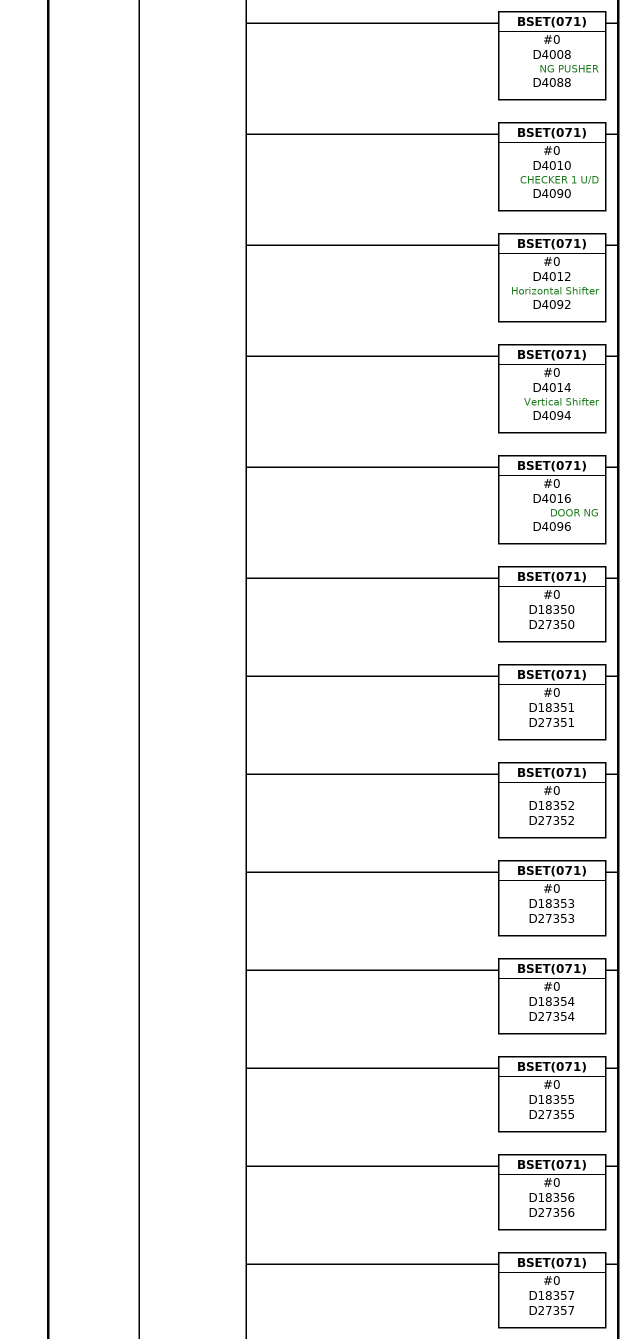
; [picture p48: Main_Control / Record, rungs 0-0]

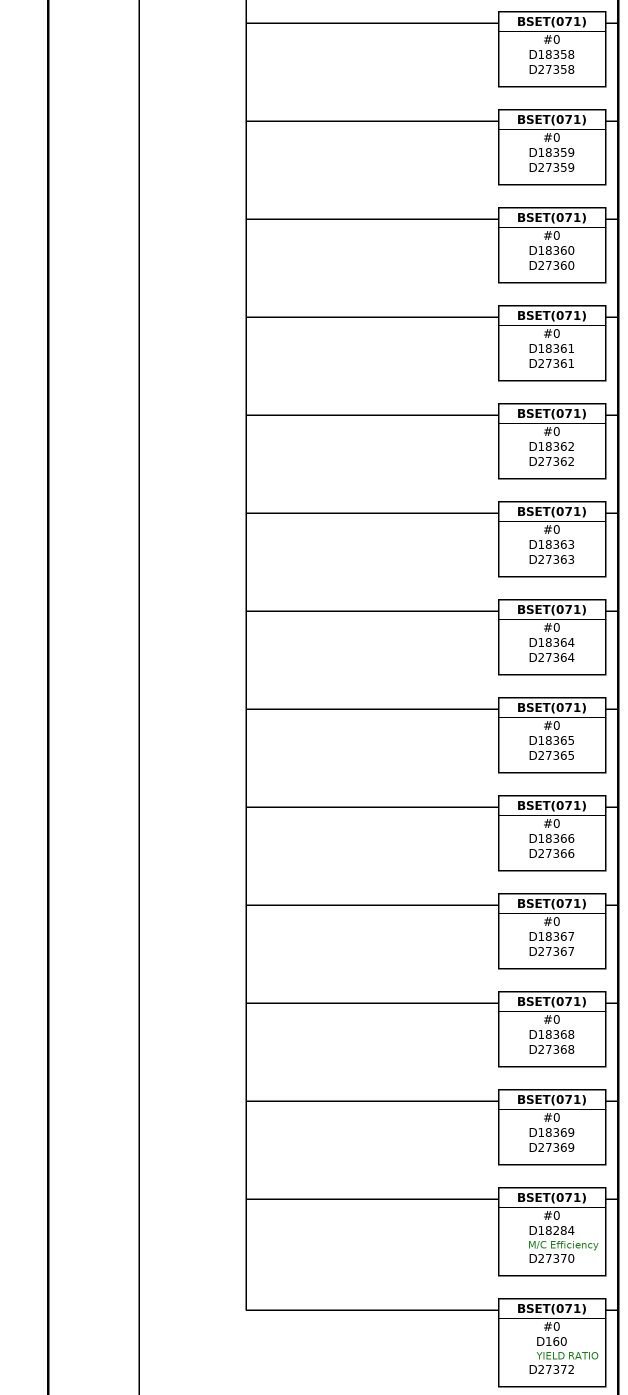

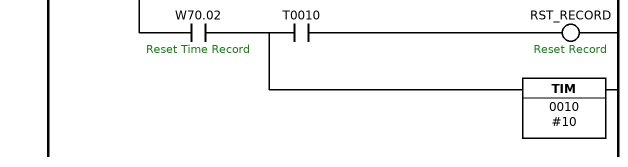
; rung 0: RESET MAIN RECORD
LD ON  ; ALWAYS ON
OUT TR0
@AND RST_RECORD  ; Reset Record
BSET(071) #0 D21300 D21399  ; OUTPUT OK
BSET(071) #0 D18251 D19299  ; M/C Cycle Time, $?St$Bk?_#[6] / $?St$Bk?_#[6]
BSET(071) #0 D19900 D19999  ; Auto Run (second), $?St$Bk?_#[7] / $?St$Bk?_#[7]
BSET(071) #0 D21100 D21199  ; STOP TIME (second)
BSET(071) #0 D21200 D21299  ; ALARM TIME (second)
BSET(071) #0 D18271 D18371  ; Input
BSET(071) #0 D20000 D20099  ; Total Alarm
BSET(071) #0 D4000 D4080  ; OVERLOAD
BSET(071) #0 D4002 D4082  ; STOPPER
BSET(071) #0 D4004 D4084  ; STOPPER CHECKER 1
BSET(071) #0 D4006 D4086  ; STOPPER CHECKER 2
BSET(071) #0 D4008 D4088  ; NG PUSHER
BSET(071) #0 D4010 D4090  ; CHECKER 1 U/D
BSET(071) #0 D4012 D4092  ; Horizontal Shifter
BSET(071) #0 D4014 D4094  ; Vertical Shifter
BSET(071) #0 D4016 D4096  ; DOOR NG
BSET(071) #0 D18350 D27350
BSET(071) #0 D18351 D27351
BSET(071) #0 D18352 D27352
BSET(071) #0 D18353 D27353
BSET(071) #0 D18354 D27354
BSET(071) #0 D18355 D27355
BSET(071) #0 D18356 D27356
BSET(071) #0 D18357 D27357
BSET(071) #0 D18358 D27358
BSET(071) #0 D18359 D27359
BSET(071) #0 D18360 D27360
BSET(071) #0 D18361 D27361
BSET(071) #0 D18362 D27362
BSET(071) #0 D18363 D27363
BSET(071) #0 D18364 D27364
BSET(071) #0 D18365 D27365
BSET(071) #0 D18366 D27366
BSET(071) #0 D18367 D27367
BSET(071) #0 D18368 D27368
BSET(071) #0 D18369 D27369
BSET(071) #0 D18284 D27370  ; M/C Efficiency
BSET(071) #0 D160 D27372  ; YIELD RATIO
LD TR0
AND W70.02  ; Reset Time Record
OUT TR0
AND T0010
OUT RST_RECORD  ; Reset Record
LD TR0
TIM 0010 #10

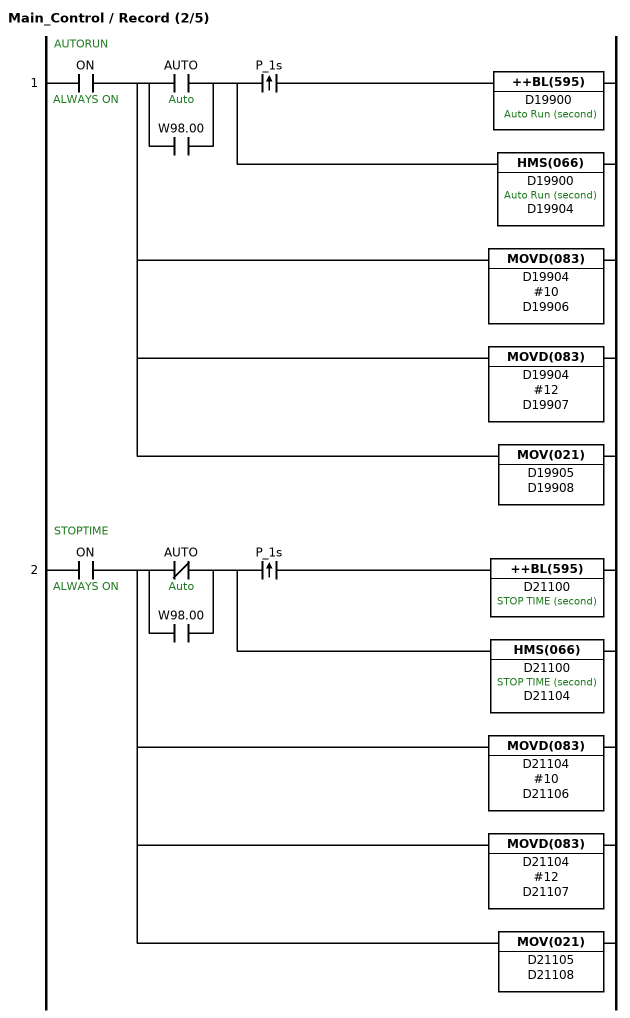
; rung 1: AUTORUN
LD ON  ; ALWAYS ON
OUT TR0
LD AUTO  ; Auto
OR W98.00
ANDLD
OUT TR1
@AND P_1s
++BL(595) D19900  ; Auto Run (second)
LD TR1
HMS(066) D19900 D19904  ; Auto Run (second)
LD TR0
MOVD(083) D19904 #10 D19906
MOVD(083) D19904 #12 D19907
MOV(021) D19905 D19908
; rung 2: STOPTIME
LD ON  ; ALWAYS ON
OUT TR0
LDNOT AUTO  ; Auto
OR W98.00
ANDLD
OUT TR1
@AND P_1s
++BL(595) D21100  ; STOP TIME (second)
LD TR1
HMS(066) D21100 D21104  ; STOP TIME (second)
LD TR0
MOVD(083) D21104 #10 D21106
MOVD(083) D21104 #12 D21107
MOV(021) D21105 D21108

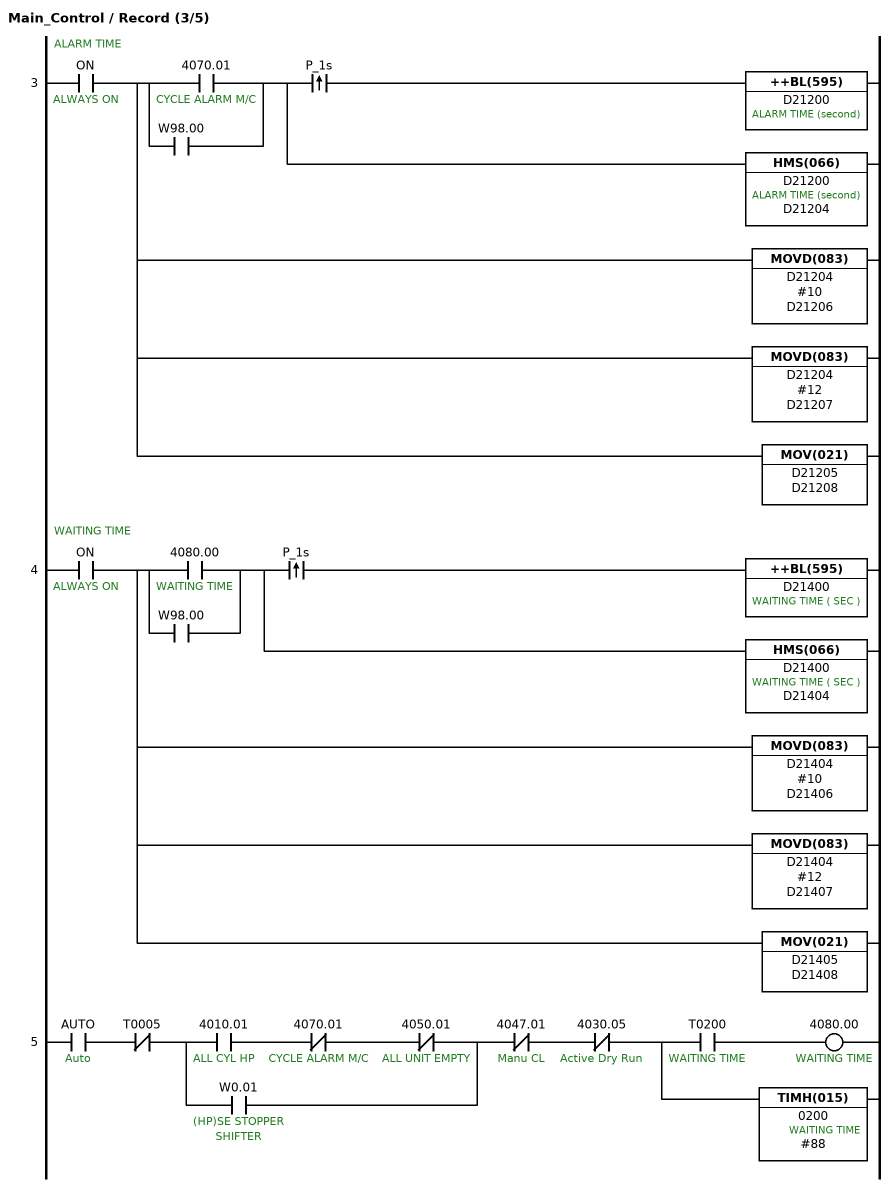
; rung 3: ALARM TIME
LD ON  ; ALWAYS ON
OUT TR0
LD 4070.01  ; CYCLE ALARM M/C
OR W98.00
ANDLD
OUT TR1
@AND P_1s
++BL(595) D21200  ; ALARM TIME (second)
LD TR1
HMS(066) D21200 D21204  ; ALARM TIME (second)
LD TR0
MOVD(083) D21204 #10 D21206
MOVD(083) D21204 #12 D21207
MOV(021) D21205 D21208
; rung 4: WAITING TIME
LD ON  ; ALWAYS ON
OUT TR0
LD 4080.00  ; WAITING TIME
OR W98.00
ANDLD
OUT TR1
@AND P_1s
++BL(595) D21400  ; WAITING TIME ( SEC )
LD TR1
HMS(066) D21400 D21404  ; WAITING TIME ( SEC )
LD TR0
MOVD(083) D21404 #10 D21406
MOVD(083) D21404 #12 D21407
MOV(021) D21405 D21408
; rung 5
LD AUTO  ; Auto
ANDNOT T0005
LD 4010.01  ; ALL CYL HP
ANDNOT 4070.01  ; CYCLE ALARM M/C
ANDNOT 4050.01  ; ALL UNIT EMPTY
OR W0.01  ; (HP)SE STOPPER SHIFTER
ANDLD
ANDNOT 4047.01  ; Manu CL
ANDNOT 4030.05  ; Active Dry Run
OUT TR0
AND T0200  ; WAITING TIME
OUT 4080.00  ; WAITING TIME
LD TR0
TIMH(015) 0200 #88  ; WAITING TIME

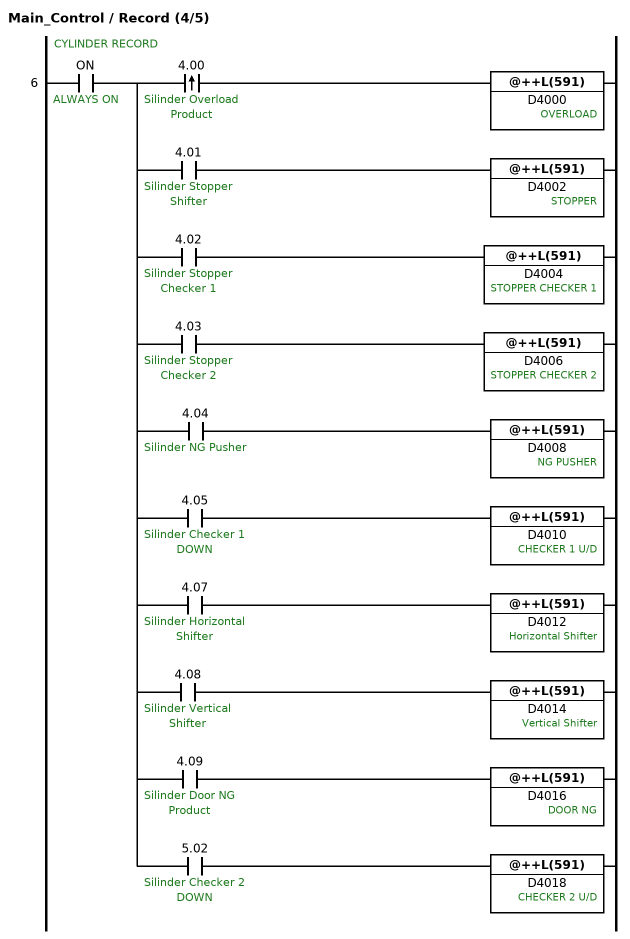
; rung 6: CYLINDER RECORD
LD ON  ; ALWAYS ON
OUT TR0
@AND 4.00  ; Silinder Overload Product
@++L(591) D4000  ; OVERLOAD
LD TR0
AND 4.01  ; Silinder Stopper Shifter
@++L(591) D4002  ; STOPPER
LD TR0
AND 4.02  ; Silinder Stopper Checker 1
@++L(591) D4004  ; STOPPER CHECKER 1
LD TR0
AND 4.03  ; Silinder Stopper Checker 2
@++L(591) D4006  ; STOPPER CHECKER 2
LD TR0
AND 4.04  ; Silinder NG Pusher
@++L(591) D4008  ; NG PUSHER
LD TR0
AND 4.05  ; Silinder Checker 1 DOWN
@++L(591) D4010  ; CHECKER 1 U/D
LD TR0
AND 4.07  ; Silinder Horizontal Shifter
@++L(591) D4012  ; Horizontal Shifter
LD TR0
AND 4.08  ; Silinder Vertical Shifter
@++L(591) D4014  ; Vertical Shifter
LD TR0
AND 4.09  ; Silinder Door NG Product
@++L(591) D4016  ; DOOR NG
LD TR0
AND 5.02  ; Silinder Checker 2 DOWN
@++L(591) D4018  ; CHECKER 2 U/D

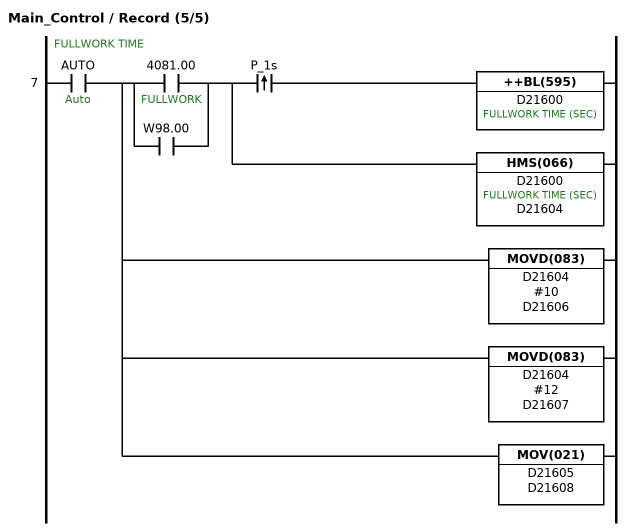
; rung 7: FULLWORK TIME
LD AUTO  ; Auto
OUT TR0
LD 4081.00  ; FULLWORK
OR W98.00
ANDLD
OUT TR1
@AND P_1s
++BL(595) D21600  ; FULLWORK TIME (SEC)
LD TR1
HMS(066) D21600 D21604  ; FULLWORK TIME (SEC)
LD TR0
MOVD(083) D21604 #10 D21606
MOVD(083) D21604 #12 D21607
MOV(021) D21605 D21608

### Section Production_Manage

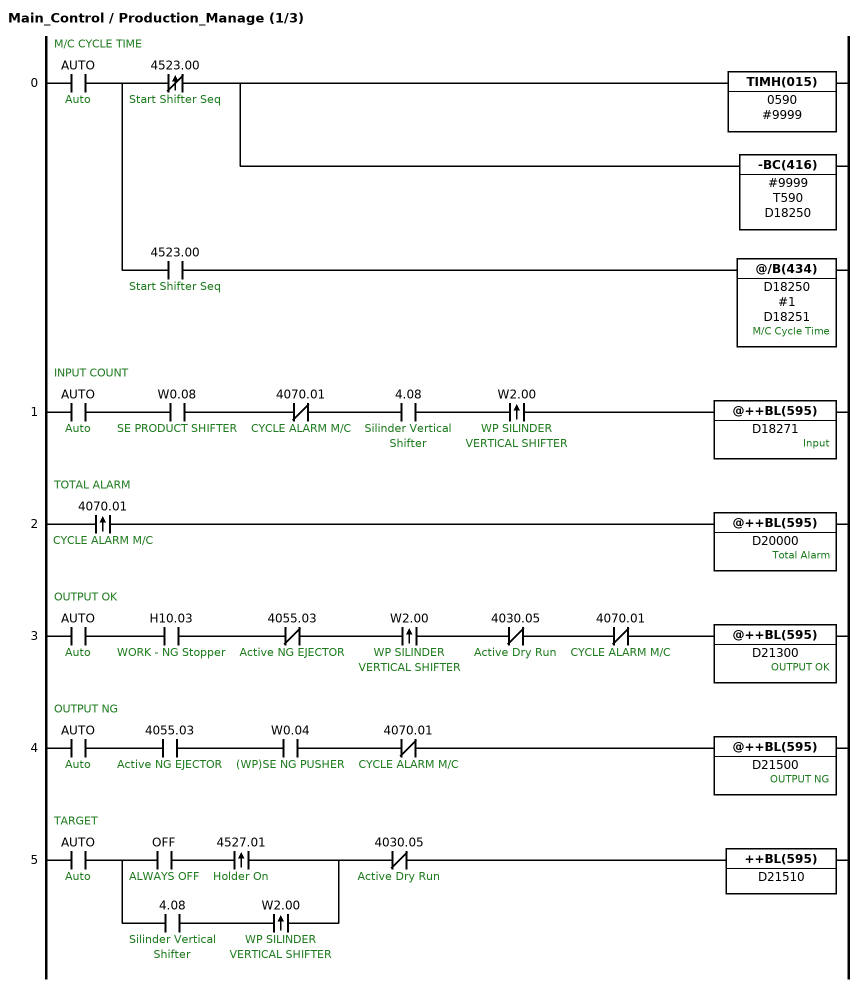
; rung 0: M/C CYCLE TIME
LD AUTO  ; Auto
OUT TR0
@ANDNOT 4523.00  ; Start Shifter Seq
TIMH(015) 0590 #9999
-BC(416) #9999 T590 D18250
LD TR0
AND 4523.00  ; Start Shifter Seq
@/B(434) D18250 #1 D18251  ; M/C Cycle Time
; rung 1: INPUT COUNT
LD AUTO  ; Auto
AND W0.08  ; SE PRODUCT SHIFTER
ANDNOT 4070.01  ; CYCLE ALARM M/C
AND 4.08  ; Silinder Vertical Shifter
@AND W2.00  ; WP SILINDER VERTICAL SHIFTER
@++BL(595) D18271  ; Input
; rung 2: TOTAL ALARM
@LD 4070.01  ; CYCLE ALARM M/C
@++BL(595) D20000  ; Total Alarm
; rung 3: OUTPUT OK
LD AUTO  ; Auto
AND H10.03  ; WORK - NG Stopper
ANDNOT 4055.03  ; Active NG EJECTOR
@AND W2.00  ; WP SILINDER VERTICAL SHIFTER
ANDNOT 4030.05  ; Active Dry Run
ANDNOT 4070.01  ; CYCLE ALARM M/C
@++BL(595) D21300  ; OUTPUT OK
; rung 4: OUTPUT NG
LD AUTO  ; Auto
AND 4055.03  ; Active NG EJECTOR
AND W0.04  ; (WP)SE NG PUSHER
ANDNOT 4070.01  ; CYCLE ALARM M/C
@++BL(595) D21500  ; OUTPUT NG
; rung 5: TARGET
LD AUTO  ; Auto
LD OFF  ; ALWAYS OFF
@AND 4527.01  ; Holder On
LD 4.08  ; Silinder Vertical Shifter
@AND W2.00  ; WP SILINDER VERTICAL SHIFTER
ORLD
ANDLD
ANDNOT 4030.05  ; Active Dry Run
++BL(595) D21510

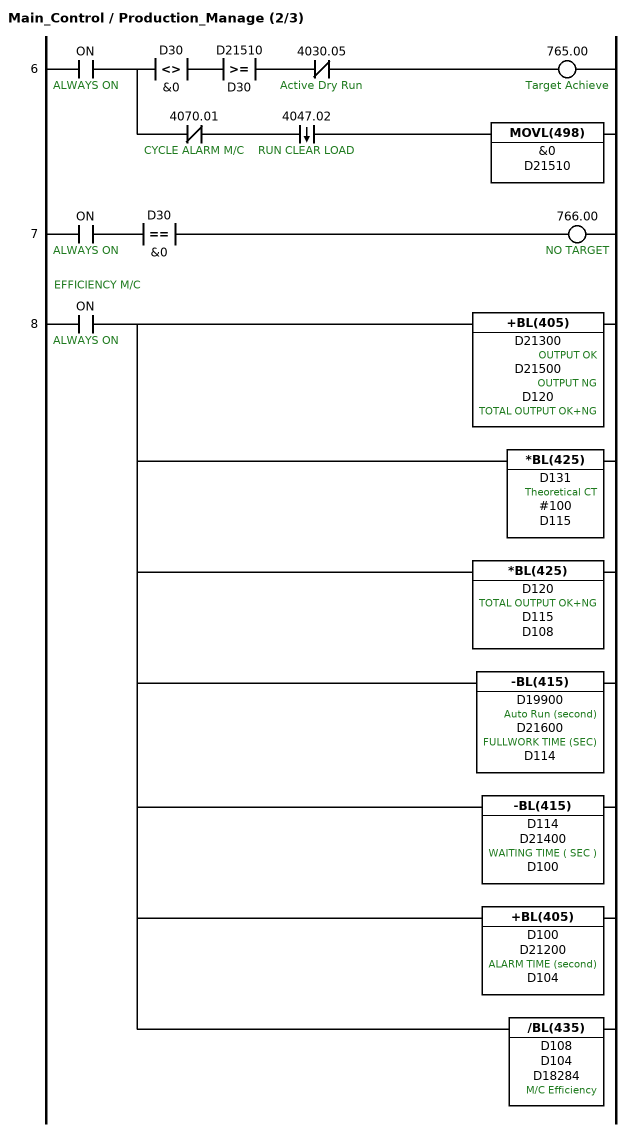
; rung 6
LD ON  ; ALWAYS ON
OUT TR0
AND<>(305) D30 &0
AND>=(325) D21510 D30
ANDNOT 4030.05  ; Active Dry Run
OUT 765.00  ; Target Achieve
LD TR0
ANDNOT 4070.01  ; CYCLE ALARM M/C
%AND 4047.02  ; RUN CLEAR LOAD
MOVL(498) &0 D21510
; rung 7
LD ON  ; ALWAYS ON
AND=(300) D30 &0
OUT 766.00  ; NO TARGET
; rung 8: EFFICIENCY M/C
LD ON  ; ALWAYS ON
+BL(405) D21300 D21500 D120  ; OUTPUT OK, OUTPUT NG, TOTAL OUTPUT OK+NG
*BL(425) D131 #100 D115  ; Theoretical CT
*BL(425) D120 D115 D108  ; TOTAL OUTPUT OK+NG
-BL(415) D19900 D21600 D114  ; Auto Run (second), FULLWORK TIME (SEC)
-BL(415) D114 D21400 D100  ; WAITING TIME ( SEC )
+BL(405) D100 D21200 D104  ; ALARM TIME (second)
/BL(435) D108 D104 D18284  ; M/C Efficiency

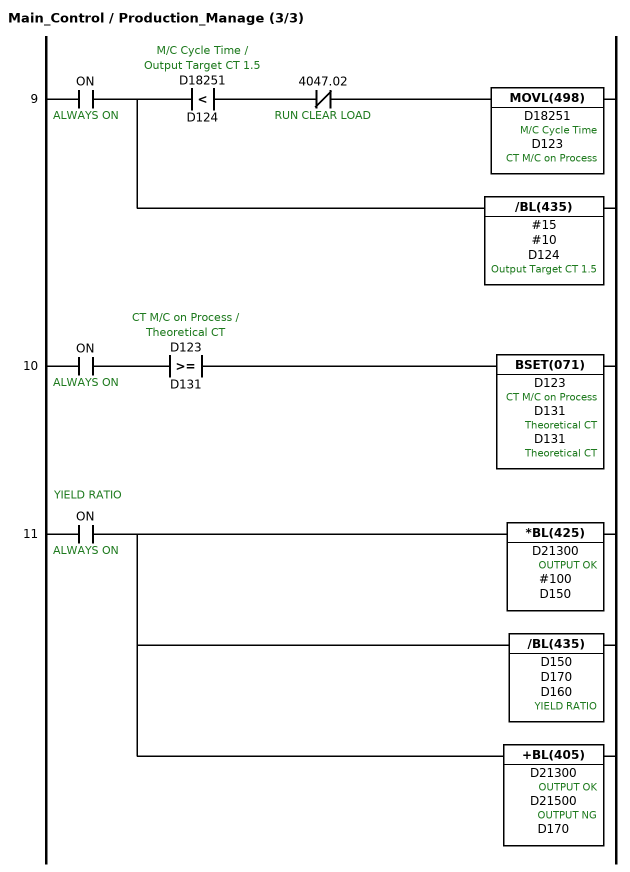
; rung 9
LD ON  ; ALWAYS ON
OUT TR0
AND<(310) D18251 D124  ; M/C Cycle Time, Output Target CT 1.5
ANDNOT 4047.02  ; RUN CLEAR LOAD
MOVL(498) D18251 D123  ; M/C Cycle Time, CT M/C on Process
LD TR0
/BL(435) #15 #10 D124  ; Output Target CT 1.5
; rung 10
LD ON  ; ALWAYS ON
AND>=(325) D123 D131  ; CT M/C on Process, Theoretical CT
BSET(071) D123 D131 D131  ; CT M/C on Process, Theoretical CT
; rung 11: YIELD RATIO
LD ON  ; ALWAYS ON
*BL(425) D21300 #100 D150  ; OUTPUT OK
/BL(435) D150 D170 D160  ; YIELD RATIO
+BL(405) D21300 D21500 D170  ; OUTPUT OK, OUTPUT NG

### Section END
; rung 0
END(001)